# EPICS alarm handler configuration: caQtDM_UnitTests/tst_qtcontrols/fixtures/alh/include_sub.alhConfig
GROUP NULL SUBROOT
CHANNEL SUBROOT sub:ch1
GROUP SUBROOT DEEP
CHANNEL DEEP sub:ch2
